// TwinCAT 3 PLC project PLCProject
// ProgramVersion: 3.1.4023.0
// libraries:
//   Tc2_Standard, * (Beckhoff Automation GmbH)
//   Tc2_System, * (Beckhoff Automation GmbH)
//   Tc3_Module, * (Beckhoff Automation GmbH)
// project tree:
//   GVLs/ GVL_Test.TcGVL
//   / PlcTask.TcTTO
//   POUs/ FB_FIFOInt.TcPOU, FB_FIFOTest.TcPOU, MAIN.TcPOU
// real-time tasks:
//   TASK PlcTask: cycle T#10ms, priority 20, ADS port 350

CONFIGURATION PLCProject
    RESOURCE PLC ON TwinCAT3
        TASK PlcTask(INTERVAL := T#10ms, PRIORITY := 20);
        PROGRAM MAIN WITH PlcTask : MAIN;
    END_RESOURCE
END_CONFIGURATION

// ---- GVLs/GVL_Test.TcGVL
{attribute 'qualified_only'}
VAR_GLOBAL
	bEnqueueItem	: BOOL;
	bDequeueItem	: BOOL;
	itemToStored	: INT;
	ExportedItem	: INT;
END_VAR

// ---- POUs/MAIN.TcPOU
PROGRAM MAIN
VAR
	fbFIFOTest : FB_FIFOTest;
END_VAR

fbFIFOTest();

END_PROGRAM

// ---- POUs/FB_FIFOTest.TcPOU
FUNCTION_BLOCK FB_FIFOTest
VAR_INPUT
END_VAR
VAR_OUTPUT
END_VAR
VAR
	fbFIFO		: FB_FIFOInt;
	
	enqTrig		: R_TRIG;
	deqTrig		: R_TRIG;
	
	bEnqueueError : BOOL;
	bDequeueError : BOOL; 
END_VAR


fbFIFO();

enqTrig(CLK := GVL_Test.bEnqueueItem);
deqTrig(CLK := GVL_Test.bDequeueItem);

IF enqTrig.Q THEN
	fbFIFO.Enqueue(i_Item := GVL_Test.itemToStored);
	bEnqueueError := fbFIFO.o_EnqueueError;
END_IF

IF deqTrig.Q THEN
	fbFIFO.Dequeue(o_Item => GVL_Test.ExportedItem);
	bDequeueError := fbFIFO.o_DequeueError;
END_IF

END_FUNCTION_BLOCK

// ---- POUs/FB_FIFOInt.TcPOU
FUNCTION_BLOCK FB_FIFOInt
VAR_INPUT
END_VAR
VAR_OUTPUT
	o_ItemCount		: INT;
	o_EnqueueError	: BOOL;
	o_DequeueError	: BOOL;
END_VAR
VAR CONSTANT
	Size 			: INT := 3;
END_VAR
VAR
	DeqOffset		: INT;
	EnqOffset		: INT;
	Items 			: ARRAY [0..Size-1] OF INT;
END_VAR

METHOD PUBLIC Dequeue : BOOL
VAR_INPUT
END_VAR
VAR_OUTPUT
	o_Item	: INT;
END_VAR

IF o_ItemCount > 0 THEN
	o_ItemCount 	:= o_ItemCount - 1;
	
	o_Item 			:= Items[DeqOffset];
	DeqOffset 		:= DeqOffset + 1;
	
	IF DeqOffset = Size THEN
		DeqOffset	:= 0;
	END_IF
	
	//Reset Enqueue error after removing an item from the array if there was an error due to attempt of overfilling
	IF o_EnqueueError THEN;
		o_EnqueueError := FALSE;
	END_IF
ELSE
	//Dequeue not possible if the item count is 0
	o_DequeueError := TRUE;
	o_Item			:= -1;
END_IF
END_METHOD

METHOD PUBLIC Enqueue : BOOL
VAR_INPUT
	i_Item	: INT;
END_VAR

IF o_ItemCount < Size THEN
	o_ItemCount 		:= o_ItemCount + 1;
	
	Items[EnqOffset] 	:= i_Item;
	EnqOffset 			:= EnqOffset + 1;
	
	IF EnqOffset = Size THEN
		EnqOffset	:= 0;
	END_IF
	
	//Reset Dequeue error after adding an item if there was an error due to having 0 items.
	IF o_DequeueError THEN;
		o_DequeueError := FALSE;
	END_IF
ELSE
	//Enqueue not possible if the item count was already equal to the buffer array size
	o_EnqueueError := TRUE;
END_IF
END_METHOD

END_FUNCTION_BLOCK
